// Mitsubishi GX Works2 project: exercicio set reset pulse   PLC: Q03UDV

PROGRAM MAIN
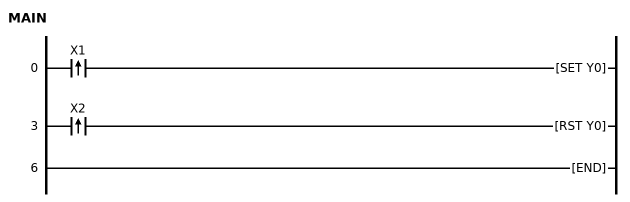
0     LDP     X1
      SET     Y0
3     LDP     X2
      RST     Y0
6     END
END_PROGRAM
